(* IEC 61131-3 sources: iec-checker/test/st, 51 files *)

(* ---- declaration-analysis.st ---- *)
(* This demo includes some declaration errors *)
TYPE
    (* String types *)
    ST0 : STRING[5];                               (* OK *)
    ST1 : STRING;                                  (* OK *)
    ST2 : STRING[5] := 'foo';                      (* OK *)
    ST3 : STRING := 'platform_dependent';          (* OK *)
    ST4 : STRING[5] := "foobar";                   (* Error *)

    (* Subrange types *)
    ANALOG_DATA1 : INT (-4095 .. 4095);          (* OK *)
    ANALOG_DATA1 : INT (-4095 .. 4095) := 2000;  (* OK *)
    ANALOG_DATA1 : INT (-4095 .. 4095) := 4095;  (* OK: See 6.4.4.4.1 *)
    ANALOG_DATA1 : INT (-4095 .. 4095) := -4095; (* OK: See 6.4.4.4.1 *)
    ANALOG_DATA2 : INT (-4095 .. 4095) := 4099;  (* Error *)
    ANALOG_DATA2 : INT (-4095 .. 4095) := -4096; (* Error *)
END_TYPE

(* ---- merge-1.st ---- *)
TYPE example_struct :
  STRUCT
    Field : BOOL;
  END_STRUCT
END_TYPE

(* ---- plcopen-cp13.st ---- *)
(* Uncompatible: Recursive functions are forbidden *)
FUNCTION Factorial : INT
    VAR_INPUT
        X : INT;
    END_VAR

    IF X > 1 THEN
        Factorial := Factorial(X - 1) * X;
    ELSE
        Factorial := X;
    END_IF;
END_FUNCTION

(* Compatible iterative implementation *)
FUNCTION Factorial_good : INT
    VAR_INPUT
        X : INT;
    END_VAR
    VAR
        Acc : INT;
    END_VAR

    FOR I := 0 TO 100 DO
        Acc := Acc * X;
    END_FOR;
    Factorial := Acc;
END_FUNCTION

(* ---- plcopen-cp4.st ---- *)
FUNCTION demo : INT
    VAR_INPUT
        x1 AT %MX40 : INT; (* PLCOPEN-CP4 *)
        x2 AT %MX41 : INT; (* PLCOPEN-CP4 *)
        x3 AT %MX510 : INT;
        w1 AT %MW10 : INT; (* adjacent words don't overlap *)
        w2 AT %MW11 : INT;
        d1 AT %MW20 : DINT; (* PLCOPEN-CP4 *)
        d2 AT %MW21 : INT; (* PLCOPEN-CP4 *)
        b1 AT %MB30 : INT; (* PLCOPEN-CP4 *)
        b2 AT %MB31 : BYTE; (* PLCOPEN-CP4 *)
        i1 AT %IW50 : INT; (* different areas don't overlap *)
        q1 AT %QW50 : INT;
        s1 AT %MW60 : INT; (* PLCOPEN-CP4 *)
        s2 AT %MW60 : INT; (* PLCOPEN-CP4 *)
    END_VAR
    x1 := 42;
END_FUNCTION

(* ---- plcopen-n4.st ---- *)
FUNCTION StartMotor : BOOL
  VAR
    goodVar : INT;
    BadVar  : INT;  (* PLCOPEN-N4 *)
  END_VAR
  StartMotor := TRUE;
END_FUNCTION

FUNCTION start_motor : BOOL    (* PLCOPEN-N4 *)
  start_motor := FALSE;
END_FUNCTION

(* ---- plcopen-n6.st ---- *)
FUNCTION Go : BOOL   (* PLCOPEN-N6 *)
  Go := TRUE;
END_FUNCTION

FUNCTION ReadAndScaleTheTemperatureInput : REAL   (* PLCOPEN-N6 *)
  ReadAndScaleTheTemperatureInput := 0.0;
END_FUNCTION

FUNCTION StartFeeding : BOOL
  StartFeeding := TRUE;
END_FUNCTION

(* ---- comparison.st ---- *)
FUNCTION_BLOCK Example
    VAR_EXTERNAL
        global_var : INT;
    END_VAR
    global_var := 42;
END_FUNCTION_BLOCK

PROGRAM Simple
  VAR_INPUT
    x : TIME;
  END_VAR
  VAR
    temp : DINT;
    i : DINT;
    arr1: ARRAY [1..2] OF BOOL;
    unused_var AT %IW1.2 : REAL := 200.0;
    head AT %B0 : INT;
  END_VAR

  IF i > 10 THEN
    temp := i;
    head := 20;
  END_IF

  WHILE i < 10 DO
    IF i = 5 THEN
      temp := i;
      EXIT;
      i := 42;
    END_IF
    i := i + 1;
  END_WHILE

  ARR1[3] := 19;
  ARR1[2,1] := 19;
  IF x = T#100MS THEN
    %B0 := 42;
  END_IF
END_PROGRAM

(* ---- cross-pou.st ---- *)
(* Programs of one task sharing outputs, globals and FB instances, directly
   and through a function block. See test_cross_pou in test_plcopen.py. *)
CONFIGURATION cfg
  VAR_GLOBAL
    gOut AT %QX2.0 : BOOL;
    gT : TON;
    g2 : INT;
    g3 : pt;
    g4 : BOOL;
    head AT %MW600 : INT;
    gm AT %MW451 : INT;
  END_VAR
  RESOURCE res ON PLC
    TASK fast(INTERVAL := T#10MS, PRIORITY := 1);
    PROGRAM i1 WITH fast : p1;
    PROGRAM i2 WITH fast : p2;
  END_RESOURCE
END_CONFIGURATION

TYPE pt : STRUCT x : INT; END_STRUCT END_TYPE

FUNCTION_BLOCK drv
  VAR_EXTERNAL gOut : BOOL; g2 : INT; gT : TON; END_VAR
  VAR_INPUT v : BOOL; END_VAR
  gOut := v;
  g2 := 1;
  gT(IN := v, PT := T#1S);
END_FUNCTION_BLOCK

PROGRAM p1
  VAR_EXTERNAL gOut : BOOL; gT : TON; g2 : INT; g3 : pt; g4 : BOOL; head : INT; END_VAR
  VAR
    out1 AT %QX0.0 : BOOL;
    r AT %MW450 : REAL;
    b1 AT %IX0.0 : BOOL;
    c : BOOL;
    t : TON;
    tmp : INT;
    d1 : drv;
    cnt : CTU;
    i : INT;
  END_VAR
  out1 := TRUE;
  gOut := c;
  gT(IN := c, PT := T#1S);
  g2 := 2;
  g3.x := 1;
  t(IN := c, PT := T#1S, Q => g4);
  %MW600 := 1;
  tmp := %MW600;
  d1(v := c);
  FOR i := 0 TO 3 DO
    cnt(CU := c);
  END_FOR;
END_PROGRAM

PROGRAM p2
  VAR_EXTERNAL gT : TON; g3 : pt; g4 : BOOL; END_VAR
  VAR
    out2 AT %QX0.0 : BOOL;
    r2 AT %MW450 : INT;
    b2 AT %IX0.0 : BOOL;
    c : BOOL;
    t : TON;
    d2 : drv;
  END_VAR
  out2 := TRUE;
  gT(IN := c, PT := T#1S);
  g3.x := 2;
  t(IN := c, PT := T#1S, Q => g4);
  d2(v := NOT c);
END_PROGRAM

(* ---- dvar.st ---- *)
FUNCTION_BLOCK Example
    VAR_EXTERNAL
        global_var : INT;
    END_VAR
    global_var := 42;
END_FUNCTION_BLOCK

PROGRAM Simple
  VAR
    temp : DINT;
    i : DINT;
    unused_var AT %IW1.2 : REAL := 200.0;
    head AT %B0 : INT;
  END_VAR

  i := head;
  i := 42;
  i := 42 + head;
  i := unused_var + 42;
  i := -head;
  i := Example(head);

END_PROGRAM

(* ---- plcopen-cp12.st ---- *)
CONFIGURATION cfg
  VAR_GLOBAL
    g_valve AT %QX1.0 : BOOL;
  END_VAR
  RESOURCE res ON PLC
    TASK main(INTERVAL := T#10MS, PRIORITY := 1);
    PROGRAM inst WITH main : demo;
  END_RESOURCE
END_CONFIGURATION

FUNCTION_BLOCK act
  VAR_OUTPUT
    out : INT;
  END_VAR
  out := 1;
END_FUNCTION_BLOCK

PROGRAM demo
  VAR_EXTERNAL
    g_valve : BOOL;
  END_VAR
  VAR
    motor AT %QW0 : INT;
    lamps AT %QW10 : WORD;
    temp : INT;
    alarm, run : BOOL;
    i : INT;
    a1 : act;
  END_VAR
  %QW1 := temp;
  IF alarm THEN
    %QW1 := 0; (* PLCOPEN-CP12 *)
  END_IF;
  IF run THEN (* exclusive branches are fine *)
    %QW3 := 1;
  ELSE
    %QW3 := 0;
  END_IF;
  motor := temp;
  %QW0 := 5; (* PLCOPEN-CP12 *)
  lamps.%X0 := TRUE; (* different bits are different outputs *)
  lamps.%X1 := TRUE;
  lamps.%X1 := FALSE; (* PLCOPEN-CP12 *)
  FOR i := 0 TO 3 DO
    %QW4 := i; (* PLCOPEN-CP12 *)
  END_FOR;
  g_valve := run;
  g_valve := alarm; (* PLCOPEN-CP12 *)
  a1(out => %QW5);
  %QW5 := 2; (* PLCOPEN-CP12 *)
  IF run THEN
    %QW6 := 1;
  ELSE
    %QW6 := 0;
  END_IF;
  %QW6 := 2; (* PLCOPEN-CP12 *)
  IF alarm THEN
    %QW7 := 0;
    RETURN;
  END_IF;
  %QW7 := 1; (* not in the same cycle as the write before RETURN *)
  temp := 1; (* not an output *)
  temp := 2;
END_PROGRAM

(* ---- plcopen-cp13-indirect.st ---- *)
FUNCTION fa : INT
  VAR_INPUT x : INT; END_VAR
  fa := fb_(x - 1); (* CP13 *)
END_FUNCTION
FUNCTION fb_ : INT
  VAR_INPUT x : INT; END_VAR
  fb_ := fa(x); (* CP13 *)
END_FUNCTION
FUNCTION fact : INT
  VAR_INPUT x : INT; END_VAR
  fact := MAX(IN1 := fact(x - 1), IN2 := 1); (* CP13 *)
END_FUNCTION
FUNCTION fact3 : INT
  VAR_INPUT x : INT; END_VAR
  fact3 := ABS(fact3(x - 1)); (* CP13 *)
END_FUNCTION
FUNCTION_BLOCK loop_fb
  VAR inner : loop_fb2; END_VAR
  inner(); (* CP13 *)
END_FUNCTION_BLOCK
FUNCTION_BLOCK loop_fb2
  VAR back : loop_fb; END_VAR
  back(); (* CP13 *)
END_FUNCTION_BLOCK
FUNCTION helper : INT
  helper := 1;
END_FUNCTION
FUNCTION user : INT
  user := helper() + helper();
END_FUNCTION

(* ---- plcopen-cp16.st ---- *)
FUNCTION_BLOCK MyFB
  VAR x : INT; END_VAR
  x := 0;
END_FUNCTION_BLOCK

FUNCTION MyFun : INT
  MyFun := 0;
END_FUNCTION

PROGRAM MyProgram
  VAR y : INT; END_VAR
  y := 0;
END_PROGRAM

(* The rule's example, after Figure 20 of IEC 61131-3 *)
PROGRAM F
  VAR_INPUT x1 : BOOL; END_VAR
  VAR_OUTPUT y1 : BOOL; END_VAR
  y1 := x1;
END_PROGRAM

PROGRAM G
  VAR_OUTPUT OUT1 : BYTE; END_VAR
  VAR FB1 : TON; FB2 : TON; END_VAR
  OUT1 := 0;
END_PROGRAM

CONFIGURATION config
  VAR_GLOBAL w : BYTE; END_VAR
  RESOURCE res1 ON PLC
    TASK Fast(INTERVAL := T#10ms, PRIORITY := 1);
    TASK Slow(INTERVAL := T#100ms, PRIORITY := 2);
    PROGRAM inst1 WITH Fast : MyProgram;
    PROGRAM inst2 WITH Slow : MyFB; (* CP16 *)
    PROGRAM inst3 : MyProgram;
    PROGRAM inst4 WITH Fast : MyFun; (* CP16 *)
    PROGRAM inst5 WITH Slow : TON; (* CP16 *)
    PROGRAM inst6 WITH Slow : Unknown;
  END_RESOURCE
  RESOURCE STATION_1 ON PROCESSOR_TYPE_1
    VAR_GLOBAL z1 : BYTE; END_VAR
    TASK SLOW_1(INTERVAL := t#20ms, PRIORITY := 2);
    TASK FAST_1(INTERVAL := t#10ms, PRIORITY := 1);
    PROGRAM P1 WITH SLOW_1 : F(x1 := %IX1.1);
    PROGRAM P2 : G(OUT1 => w,
      FB1 WITH SLOW_1, (* CP16 *)
      FB2 WITH FAST_1); (* CP16 *)
  END_RESOURCE
END_CONFIGURATION

(* ---- plcopen-cp17-members.st ---- *)
TYPE pt : STRUCT x : INT; y : INT; END_STRUCT END_TYPE
FUNCTION_BLOCK f
  VAR_INPUT
    pin : pt;
    other : pt;
  END_VAR
  VAR_OUTPUT
    pout : pt;
    q : INT;
  END_VAR
  pout.x := pin.x;
  other.x := 1;
  q := other.y;
END_FUNCTION_BLOCK

(* ---- plcopen-cp17.st ---- *)
FUNCTION_BLOCK FB_CP17_Test
VAR_INPUT
    in_ok_read_only       : INT;   // Compliant: read at least once, never written
    in_violate_unused     : INT;   // Violation: never read
    in_violate_write_only : INT;   // Violation: written, not read
    in_violate_read_write : INT;   // Violation: read but also written

    idx_read_only           : INT;   // Compliant: only read as array index
    idx_violate_write_only  : INT;   // Violation: written, not read
    func_violate_unused     : INT;   // Violation: never use
    func_read_only          : INT;   // Compliant: only read in func call
    func_violate_write      : INT;   // Violation: written in func call
END_VAR

VAR_OUTPUT
    out_ok_written        : INT;   // Compliant: written at least once
    out_violate_unused    : INT;   // Violation: never written
    out_violate_read_only : INT;   // Violation: read but not written
END_VAR

VAR_IN_OUT
    io_ok_read_only       : INT;   // Compliant: read only
    io_ok_write_only      : INT;   // Compliant: written only
    io_ok_read_write      : INT;   // Compliant: both read and written
    io_violate_unused     : INT;   // Violation: neither read nor written
END_VAR

VAR
    temp : INT;
    arr  : ARRAY[0..9] OF INT;
    func : MYFUNC;
END_VAR

(* ===== VAR_INPUT tests ===== *)

(* Compliant: input parameter is read *)
temp := in_ok_read_only + 1;

(* Violation: in_violate_unused is never used *)

(* Violation: input parameter is written *)
in_violate_write_only := 100;

(* Violation: input parameter is both read and written *)
temp := in_violate_read_write;
in_violate_read_write := temp + 1;

(* ===== VAR_OUTPUT tests ===== *)

(* Compliant: output parameter is written *)
out_ok_written := temp;

(* Violation: out_violate_unused is never written *)

(* Violation: output parameter is read but not written *)
temp := out_violate_read_only;

(* ===== VAR_IN_OUT tests ===== *)

(* Compliant: read only *)
temp := temp + io_ok_read_only;

(* Compliant: written only *)
io_ok_write_only := 10;

(* Compliant: both read and written *)
io_ok_read_write := io_ok_read_write + 1;

(* Violation: io_violate_unused is never used *)

(* ===== special tests for LHS handling ===== *)

(* Important case:
   idx_read_only is used only to locate the write target arr[idx_read_only].
   It should be counted as READ, not WRITE.
   However, *)
arr[idx_read_only] := 5;

(* Violation:
   idx_violate_write_only is written, but never read. *)
idx_violate_write_only := 3;

(* Function Call *)
func(func_violate_unused := func_read_only, func_violate_unused => func_violate_write);

END_FUNCTION_BLOCK

(*
 * The reported result should be:
 * 1. in_violate_unused => should be read
 * 2. in_violate_write_only => should not be written, should be read (2 * warnings reported)
 * 3. in_violate_read_write => should not be written
 * 4. out_violate_unused => should be written
 * 5. out_violate_read_only => should be written
 * 6. io_violate_unused => should be written/read
 * 7. idx_violate_write_only => should not be written, should be read (2 * warnings reported)
 * 8. func_violate_unused => never used, should be read
 * 9. func_violate_write => should not be written, should be read (2 * warnings reported)
*)

(* ---- plcopen-cp2-library.st ---- *)
(* A library: no program uses these here, but applications do. *)
FUNCTION Scale : INT
  VAR_INPUT x : INT; END_VAR
  Scale := x * 2;
END_FUNCTION

FUNCTION_BLOCK Valve
  VAR_OUTPUT open : BOOL; END_VAR
  open := TRUE;
END_FUNCTION_BLOCK

(* ---- plcopen-cp2-unreferenced.st ---- *)
CONFIGURATION cfg
  VAR_GLOBAL
    g_valve : Valve;
  END_VAR
  RESOURCE res ON PLC
    TASK t (INTERVAL := T#10ms, PRIORITY := 1);
    PROGRAM main_inst WITH t : Main;
  END_RESOURCE
END_CONFIGURATION

FUNCTION Scale : INT
  VAR_INPUT x : INT; END_VAR
  Scale := x * 2;
END_FUNCTION

FUNCTION Clamp : INT
  VAR_INPUT x : INT; END_VAR
  Clamp := x;
END_FUNCTION

FUNCTION Unused : INT (* CP2 *)
  VAR_INPUT x : INT; END_VAR
  Unused := x;
END_FUNCTION

FUNCTION Recurse : INT (* CP2 *)
  VAR_INPUT n : INT; END_VAR
  Recurse := Recurse(n - 1);
END_FUNCTION

FUNCTION OnlyForDeadFb : INT (* CP2 *)
  OnlyForDeadFb := 1;
END_FUNCTION

FUNCTION_BLOCK Valve
  VAR_OUTPUT open : BOOL; END_VAR
  open := TRUE;
END_FUNCTION_BLOCK

FUNCTION_BLOCK Pump
  VAR_OUTPUT running : BOOL; END_VAR
  running := TRUE;
END_FUNCTION_BLOCK

FUNCTION_BLOCK Mixer
  VAR_OUTPUT active : BOOL; END_VAR
  active := TRUE;
END_FUNCTION_BLOCK

FUNCTION_BLOCK DeadFb (* CP2 *)
  VAR_OUTPUT v : INT; END_VAR
  v := OnlyForDeadFb();
END_FUNCTION_BLOCK

TYPE Station :
  STRUCT
    mixer : Mixer;
  END_STRUCT;
END_TYPE

PROGRAM Main
  VAR
    pumps : ARRAY [1..2] OF Pump;
    st : Station;
    y : INT;
  END_VAR
  y := Clamp(Scale(y));
END_PROGRAM

PROGRAM Spare (* CP2 *)
  VAR y : INT; END_VAR
  y := 1;
END_PROGRAM

(* ---- plcopen-cp20.st ---- *)
FUNCTION_BLOCK counter
  VAR_INPUT
    x : BOOL;
  END_VAR
  VAR_OUTPUT
    n : INT;
  END_VAR
  IF x THEN
    n := n + 1;
  END_IF;
END_FUNCTION_BLOCK

FUNCTION helper : INT
  VAR_INPUT
    a : INT;
  END_VAR
  helper := a;
END_FUNCTION

PROGRAM demo
  VAR
    edge1, edge2 : R_TRIG;
    t1 : TON;
    c1 : counter;
    input_a, input_b, run : BOOL;
    i, y : INT;
  END_VAR
  edge1(CLK := input_a);
  edge1(CLK := input_b); (* PLCOPEN-CP20 *)
  edge2(CLK := input_a); (* a different instance *)
  IF run THEN (* exclusive branches are fine *)
    t1(IN := TRUE, PT := T#1S);
  ELSE
    t1(IN := FALSE, PT := T#1S);
  END_IF;
  FOR i := 0 TO 3 DO
    c1(x := run); (* PLCOPEN-CP20 *)
  END_FOR;
  helper(a := 1); (* functions can be called any number of times *)
  helper(a := 2);
  y := helper(3);
END_PROGRAM

(* ---- plcopen-cp25.st ---- *)
TYPE percent : USINT; END_TYPE

TYPE motor_t :
  STRUCT
    speed : DINT;
    temp : REAL;
  END_STRUCT
END_TYPE

FUNCTION_BLOCK sensor
  VAR_INPUT
    limit : INT;
  END_VAR
  VAR_OUTPUT
    value : LREAL;
  END_VAR
  value := 1.0;
END_FUNCTION_BLOCK

FUNCTION scale : DINT
  VAR_INPUT
    x : INT;
    k : REAL;
  END_VAR
  scale := x;
END_FUNCTION

PROGRAM demo
  VAR
    s : SINT;
    I : INT := 10;
    J : REAL := 0.55;
    d : DINT;
    u : UINT;
    lr : LREAL;
    p : percent;
    m : motor_t;
    arr : ARRAY [0..3] OF DINT;
    fb : sensor;
    c : BOOL;
  END_VAR
  (* Conversions without loss are allowed (Table 11) *)
  I := s;
  d := I;
  J := I;
  lr := J;
  c := I < J;
  (* Explicit conversions *)
  I := REAL_TO_INT(J);
  J := INT_TO_REAL(I);
  I := DINT_TO_INT(d);
  (* Lossy implicit conversions *)
  I := J; (* PLCOPEN-CP25 *)
  I := I * J; (* PLCOPEN-CP25 *)
  I := d; (* PLCOPEN-CP25 *)
  I := d + 1; (* PLCOPEN-CP25 *)
  u := I; (* PLCOPEN-CP25 *)
  J := lr; (* PLCOPEN-CP25 *)
  I := 5.7; (* PLCOPEN-CP25 *)
  s := 300; (* PLCOPEN-CP25 *)
  s := 100;
  u := -1; (* PLCOPEN-CP25 *)
  p := I; (* PLCOPEN-CP25 *)
  I := m.speed; (* PLCOPEN-CP25 *)
  I := arr[1]; (* PLCOPEN-CP25 *)
  J := fb.value; (* PLCOPEN-CP25 *)
  I := scale(I, J); (* PLCOPEN-CP25 *)
  I := %IW0; (* PLCOPEN-CP25 *)
  d := %IW0;
  (* Operands without a lossless common type *)
  c := d < J; (* PLCOPEN-CP25 *)
  c := I = u; (* PLCOPEN-CP25 *)
  (* Arguments *)
  fb(limit := d); (* PLCOPEN-CP25 *)
  fb(limit := I);
  d := scale(d, J); (* PLCOPEN-CP25 *)
  d := scale(x := I, k := lr); (* PLCOPEN-CP25 *)
END_PROGRAM

(* ---- plcopen-cp28.st ---- *)
PROGRAM demo
    VAR
        x : TIME;
        y : TIME;
        t1 : TON;
        now, shift_start : TOD;
        today, due : DATE;
        ready, b : BOOL;
    END_VAR

    IF x = T#100MS THEN (* PLCOPEN CP-28 *)
      x := x + 1;
    END_IF;

    IF x <> T#100MS THEN (* PLCOPEN CP-28 *)
      x := x + 1;
    END_IF;

    IF T#100MS = x THEN (* PLCOPEN CP-28 *)
      x := x + 1;
    END_IF;

    IF T#100MS <> x THEN (* PLCOPEN CP-28 *)
      x := x + 1;
    END_IF;

    IF REAL_TO_INT(x) <> 0 THEN (* PLCOPEN CP-28: a time in an integer *)
      x := x + 1;
    END_IF;

    IF x = y THEN (* PLCOPEN CP-28 *)
      x := T#0S;
    END_IF;
    IF t1.ET = x THEN (* PLCOPEN CP-28 *)
      x := T#0S;
    END_IF;
    b := ready AND x <> y; (* PLCOPEN CP-28 *)
    IF now = shift_start THEN (* PLCOPEN CP-28 *)
      x := T#0S;
    END_IF;
    IF today = due THEN (* dates can be compared for equality *)
      x := T#0S;
    END_IF;
    IF t1.ET >= x THEN (* ordering comparisons are fine *)
      x := T#0S;
    END_IF;
    IF today = D#2024-01-01 THEN (* date literals are dates *)
      x := T#0S;
    END_IF;
    IF now = TOD#08:00:00 THEN (* PLCOPEN CP-28 *)
      x := T#0S;
    END_IF;
END_PROGRAM

FUNCTION_BLOCK Stopwatch
    VAR_INPUT run : BOOL; END_VAR
    VAR_OUTPUT elapsed_ms : DINT; count : INT; END_VAR
    VAR t : TON; END_VAR
    t(IN := run, PT := T#1H);
    elapsed_ms := TIME_TO_DINT(t.ET);
    count := count + 1;
END_FUNCTION_BLOCK

FUNCTION SecondsOf : DINT
    VAR_INPUT d : TIME; END_VAR
    SecondsOf := TIME_TO_DINT(d) / 1000;
END_FUNCTION

PROGRAM integers
    VAR
        t1 : TON;
        sw : Stopwatch;
        ms, secs, n, code : DINT;
        r : REAL;
    END_VAR
    (* The rule's example: a time in integer format. *)
    IF TIME_TO_DINT(t1.ET) = 10000 THEN (* PLCOPEN CP-28 *)
      n := 0;
    END_IF;
    ms := TIME_TO_DINT(t1.ET);
    secs := ms / 1000;
    IF secs = 10 THEN (* PLCOPEN CP-28 *)
      n := 0;
    END_IF;
    IF TO_DINT(t1.ET) <> ms THEN (* PLCOPEN CP-28 *)
      n := 0;
    END_IF;
    IF sw.elapsed_ms = 500 THEN (* PLCOPEN CP-28 *)
      n := 0;
    END_IF;
    IF SecondsOf(t1.ET) = 3 THEN (* PLCOPEN CP-28 *)
      n := 0;
    END_IF;
    IF ms > 10000 THEN (* ordering comparisons are fine *)
      n := 0;
    END_IF;
    IF sw.count = 3 OR code = 7 THEN (* other integers are fine *)
      n := 0;
    END_IF;
    r := TIME_TO_REAL(t1.ET);
    IF n = 0 THEN
      n := 1;
    END_IF;
END_PROGRAM

(* ---- plcopen-cp6-constants.st ---- *)
CONFIGURATION cfg
  VAR_GLOBAL CONSTANT
    MAX_SPEED : INT := 1500;
  END_VAR
  VAR_GLOBAL
    ModeAuto : BOOL;
  END_VAR
END_CONFIGURATION

FUNCTION_BLOCK motor
  VAR_EXTERNAL CONSTANT
    MAX_SPEED : INT;
  END_VAR
  VAR_EXTERNAL
    ModeAuto : BOOL; (* CP6 *)
  END_VAR
  VAR_OUTPUT q : BOOL; END_VAR
  q := ModeAuto AND MAX_SPEED > 0;
END_FUNCTION_BLOCK

FUNCTION limit_of : INT
  VAR_EXTERNAL
    MAX_SPEED : INT; (* references a constant global *)
  END_VAR
  limit_of := MAX_SPEED;
END_FUNCTION

(* ---- plcopen-cp6.st ---- *)
FUNCTION demo : INT
    VAR_EXTERNAL
        x1 : INT; (* PLCOPEN-CP6 *)
    END_VAR
    x1 := 42;
END_FUNCTION

FUNCTION_BLOCK demo
    VAR_EXTERNAL
        x1 : INT; (* PLCOPEN-CP6 *)
    END_VAR
    x1 := 42;
END_FUNCTION_BLOCK

PROGRAM demo
    VAR_EXTERNAL
        x1 : INT;
    END_VAR
    x1 := 42;
END_PROGRAM

CLASS test1
  VAR_EXTERNAL
    x1 : INT; (* PLCOPEN-CP6 *)
  END_VAR

  METHOD PRIVATE count
    x1 := 42;
  END_METHOD

END_CLASS

(* ---- plcopen-cp7.st ---- *)
FUNCTION_BLOCK Scaler
  VAR_INPUT P1 : INT; P2 : INT; END_VAR
  VAR_OUTPUT Out : INT; xError : BOOL; iError : INT; END_VAR
  Out := P1 * P2;
  xError := FALSE;
  iError := 0;
END_FUNCTION_BLOCK

FUNCTION ReadSensor : INT
  VAR_INPUT channel : INT; END_VAR
  VAR_OUTPUT ErrorCode : INT; END_VAR
  ReadSensor := channel;
  ErrorCode := 0;
END_FUNCTION

FUNCTION_BLOCK Wrapper
  VAR_OUTPUT xError : BOOL; END_VAR
  VAR inner : Scaler; END_VAR
  inner(P1 := 1, P2 := 2, xError => xError);   (* passed on as its own output *)
END_FUNCTION_BLOCK

PROGRAM Main
  VAR
    Cond : BOOL;
    Eff1 : INT;
    Eff2 : INT;
    Result : INT;
    CriticalThreshold : INT;
    instance : Scaler;
    checked : Scaler;
    connected : Scaler;
    ignored : Scaler;
    err : BOOL;
    code : INT;
    unread : INT;
    unreadFlag : BOOL;
    value : INT;
    move : MC_MoveAbsolute;
    power : MC_Power;
    wrap : Wrapper;
  END_VAR
  (* The rule's example: Result is used without checking the error *)
  instance(P1 := Eff1, P2 := Eff2);   (* PLCOPEN-CP7 *)
  Result := instance.Out;
  CriticalThreshold := Result + 10000;

  (* Tested: read directly, or connected and read *)
  checked(P1 := Eff1, P2 := Eff2);
  IF NOT checked.xError AND checked.iError = 0 THEN
    CriticalThreshold := checked.Out + 10000;
  END_IF;
  connected(P1 := Eff1, P2 := Eff2, xError => err, iError => code);
  IF NOT err AND code = 0 THEN
    Result := connected.Out;
  END_IF;
  ignored(P1 := 1, P2 := 2, xError => unreadFlag, iError => unread);   (* PLCOPEN-CP7 *)

  (* Functions with an error output *)
  value := ReadSensor(channel := 1, ErrorCode => code);
  value := ReadSensor(channel := 2);   (* PLCOPEN-CP7 *)
  unread := ReadSensor(channel := 3, ErrorCode => unread);   (* PLCOPEN-CP7 *)

  (* Motion control blocks *)
  move(Execute := Cond);   (* PLCOPEN-CP7 *)
  power(Enable := TRUE);
  IF power.Error THEN
    Cond := FALSE;
  END_IF;   (* testing Error is enough *)

  (* The error of wrap is passed on as its own output *)
  wrap();
  Cond := wrap.xError;
END_PROGRAM

(* ---- plcopen-cp9.st ---- *)
(* Example from PLCOpen guidelines, page 60.

   The following Function block CHARCURVE has:
   Number of Statements 18
   McCabe complexity of 12
   Prater complexity of 3,89
   Halstead complexity of 44,9
   Elshof complexity of 0,14

  Counting each statement once, including ELSIF but not ELSE, gives their 18
  statements. Their McCabe value comes out with the "plcopen" variant; the
  standard McCabe complexity is 8. CHARCURVE2 is the improved version of the
  rule's example: 12 statements, and McCabe complexity 8 (standard: 6).
 *)

FUNCTION_BLOCK CHARCURVE
  VAR_INPUT
    IN:INT;
    N:BYTE;
  END_VAR
  (* VAR_IN_OUT *)
    (* P : ARRAY [0 .. 10] OF POINT; *)
  (* END_VAR *)
  VAR_OUTPUT
    OUT:INT;
    ERR: BYTE;
  END_VAR
  VAR
    I:INT;
  END_VAR

  IF N > 1 AND N < 12 THEN
    ERR:=0;
    (* IF IN < P[0].X THEN *)
    IF IN < a THEN
      ERR := 2;
      OUT := DINT_TO_INT(a);
    (* ELSIF IN > P[N-1].X THEN *)
    ELSIF IN > a THEN
      ERR := 2;
      OUT := DINT_TO_INT(a);
    ELSE
      FOR I:=1 TO N-1 DO
        (* IF P[I-1].X >= P[I].X THEN *)
        IF a >= a THEN
          ERR:=1;
          EXIT;
        END_IF;
        (* IF IN <= P[I].X THEN *)
        IF IN <= a THEN
          EXIT;
        END_IF;
      END_FOR;
      IF ERR = 0 THEN
        (* OUT := DINT_TO_INT(P[I].Y - (P[I].X-IN) * (P[I].Y-P[I-1].Y) / (P[I].X-P[I-1].X)); *)
        OUT := DINT_TO_INT(a - (a - IN) * (a - a) / (a - a));
      ELSE
        OUT:=0;
      END_IF;
    END_IF;
  ELSE
    ERR := 4;
  END_IF;
END_FUNCTION_BLOCK

FUNCTION_BLOCK CHARCURVE2
  VAR_INPUT
    IN:INT;
    N:BYTE;
  END_VAR
  VAR_OUTPUT
    OUT:INT;
    ERR: BYTE;
  END_VAR
  VAR
    I:INT;
    iIndexFound:INT;
  END_VAR

  OUT := 0;
  ERR := 0;
  iIndexFound := -1;
  FOR I := 1 TO N-1 DO
    (* IF iIndexFound < 0 AND ERR = 0 THEN *)
    IF iIndexFound < 0 AND ERR = 0 THEN
      (* IF P[I-1].X >= P[I].X THEN *)
      IF a >= a THEN
        ERR := 1;
      (* ELSIF IN <= P[I].X THEN *)
      ELSIF IN <= a THEN
        iIndexFound := I;
      END_IF;
    END_IF;
  END_FOR;
  IF ERR = 0 THEN
    (* OUT := CalculateOut(P[iIndexFound], P[iIndexFound - 1]); *)
    OUT := a;
  ELSE
    OUT := 0;
  END_IF;
END_FUNCTION_BLOCK

(* ---- plcopen-l22.st ---- *)
FUNCTION_BLOCK Stepper
  VAR_INPUT step : INT; END_VAR
  VAR_IN_OUT pos : INT; END_VAR
  VAR_OUTPUT next : INT; END_VAR
  pos := pos + step;
  next := pos;
END_FUNCTION_BLOCK

FUNCTION Bump : INT
  VAR_IN_OUT x : INT; END_VAR
  x := x + 1;
  Bump := x;
END_FUNCTION

PROGRAM l22
  VAR
    i : INT := 0;
    j : INT := 0;
    n : INT := 10;
    k : INT := 1;
    arr : ARRAY[0..10] OF INT;
    cfg : Limits;
    st : Stepper;
  END_VAR

  (* Case 1: Direct assignment in body — violation *)
  FOR i := 0 TO 10 BY 2 DO
    IF arr[i] = 42 THEN
      i := 10; (* L22 *)
    END_IF;
  END_FOR;

  (* Case 2: No violation — different variable *)
  FOR i := 0 TO 10 DO
    j := i + 1;
  END_FOR;

  (* Case 3: Nested FOR — inner loop modifies outer var — violation *)
  FOR i := 0 TO 10 DO
    FOR j := 0 TO 5 DO
      i := j; (* L22 *)
    END_FOR;
  END_FOR;

  (* Case 4: Nested FOR — inner loop modifies its own var — violation *)
  FOR i := 0 TO 10 DO
    FOR j := 0 TO 5 DO
      j := 0; (* L22 *)
    END_FOR;
  END_FOR;

  (* Case 5: Nested FOR reuses the outer control variable *)
  FOR i := 0 TO 10 DO
    FOR i := 0 TO 5 DO (* L22 *)
      j := i;
    END_FOR;
  END_FOR;

  (* Case 6: Written through an output and a VAR_IN_OUT *)
  FOR i := 0 TO 10 DO
    st(step := 1, pos := i, next => j); (* L22 *)
  END_FOR;
  FOR j := 0 TO 10 DO
    st(step := 1, pos := k, next => j); (* L22 *)
  END_FOR;
  FOR i := 0 TO 10 DO
    j := Bump(i); (* L22 *)
  END_FOR;

  (* Case 7: The final value and increment change *)
  FOR i := 0 TO n BY k DO
    n := n - 1; (* L22 *)
    k := 2; (* L22 *)
  END_FOR;
  FOR i := 0 TO cfg.max DO
    cfg.max := 5; (* L22 *)
    cfg.min := 1;
  END_FOR;
  FOR i := 0 TO arr[j] DO
    j := j + 1; (* L22 *)
  END_FOR;

  (* Case 8: The initial value is evaluated once *)
  FOR i := j TO 10 DO
    j := 0;
  END_FOR;
END_PROGRAM

(* ---- plcopen-n10-kinds.st ---- *)
TYPE EColor : (Red, Green); END_TYPE
TYPE Error : (Minor, Major); END_TYPE   (* PLCOPEN-N10 *)
TYPE EN_Level : INT (Low := 1, High := 2); END_TYPE
TYPE ELevel : INT (Low2 := 1, High2 := 2); END_TYPE   (* PLCOPEN-N10 *)
TYPE STPoint : STRUCT x : INT; END_STRUCT; END_TYPE
TYPE T_Speed : REAL; END_TYPE
TYPE Speed2 : REAL; END_TYPE   (* PLCOPEN-N10 *)

FUNCTION FUScale : INT
  FUScale := 1;
END_FUNCTION

FUNCTION Scale : INT   (* PLCOPEN-N10 *)
  Scale := 1;
END_FUNCTION

FUNCTION_BLOCK FBPump
  VAR x : INT; END_VAR
  x := 1;
END_FUNCTION_BLOCK

FUNCTION_BLOCK FBpump2   (* PLCOPEN-N10 *)
  VAR x : INT; END_VAR
  x := 1;
END_FUNCTION_BLOCK

PROGRAM PRGMain
  VAR x : INT; END_VAR
  x := 1;
END_PROGRAM

PROGRAM Main   (* PLCOPEN-N10 *)
  VAR x : INT; END_VAR
  x := 1;
END_PROGRAM

(* ---- plcopen-n10.st ---- *)
TYPE
  Color : (Red, Green, Blue);   (* PLCOPEN-N10 *)
END_TYPE

TYPE
  E_Direction : (North, South, East, West);
END_TYPE

FUNCTION_BLOCK Motor   (* PLCOPEN-N10 *)
  VAR
    speed : INT;
  END_VAR
  speed := 0;
END_FUNCTION_BLOCK

FUNCTION_BLOCK FB_Pump
  VAR
    flow : REAL;
  END_VAR
  flow := 0.0;
END_FUNCTION_BLOCK

(* ---- plcopen-n2-scopes.st ---- *)
TYPE Point : STRUCT x : INT; y : INT; END_STRUCT; END_TYPE
TYPE Mode : (Auto, Manual); END_TYPE
TYPE Temperature : REAL; END_TYPE
TYPE Counter : INT; END_TYPE

FUNCTION_BLOCK Pump
  VAR_INPUT
    pxEnable : BOOL;
    xEnable : BOOL;         (* PLCOPEN-N2 *)
  END_VAR
  VAR_OUTPUT
    piCount : INT;
  END_VAR
  VAR
    xReady : BOOL;
    x_done : BOOL;
    xylophone : BOOL;       (* PLCOPEN-N2 *)
    index : INT;            (* PLCOPEN-N2 *)
    todStart : TIME_OF_DAY;
    todEnd : TOD;
    StartAt : TOD;          (* PLCOPEN-N2 *)
    aValues : ARRAY [0..3] OF INT;
    values : ARRAY [0..3] OF INT;  (* PLCOPEN-N2 *)
    stOrigin : Point;
    origin : Point;         (* PLCOPEN-N2 *)
    eMode : Mode;
    mode : Mode;            (* PLCOPEN-N2 *)
    fbTimer : TON;
    timer : TON;            (* PLCOPEN-N2 *)
    tempOven : Temperature;
    oven : Temperature;     (* PLCOPEN-N2 *)
    iTotal : Counter;
    total : Counter;        (* PLCOPEN-N2 *)
    unknown : SomeType;
  END_VAR
  xReady := pxEnable;
END_FUNCTION_BLOCK

PROGRAM Main
  VAR xOn : BOOL; END_VAR
  xOn := TRUE;
END_PROGRAM

CONFIGURATION cfg
  VAR_GLOBAL
    gxRunning : BOOL;
    xStopped : BOOL;        (* PLCOPEN-N2 *)
    gCount : INT;           (* PLCOPEN-N2 *)
  END_VAR
  RESOURCE res ON PLC
    VAR_GLOBAL
      giLevel : INT;
      level : INT;          (* PLCOPEN-N2 *)
    END_VAR
    TASK main(INTERVAL := T#10ms, PRIORITY := 1);
    PROGRAM inst WITH main : Main;
  END_RESOURCE
END_CONFIGURATION

(* ---- plcopen-n3-names.st ---- *)
TYPE MAX : STRUCT TP : INT; y : INT; END_STRUCT END_TYPE
TYPE mode : (SEL, RUNNING); END_TYPE
FUNCTION_BLOCK TON2
VAR LEFT, LIMIT, LOG, LE, Temp : INT; END_VAR
LEFT := 1;
END_FUNCTION_BLOCK
FUNCTION LEN : INT
LEN := 1;
END_FUNCTION
PROGRAM CTUD
VAR x : INT; END_VAR
x := 1;
END_PROGRAM

(* ---- plcopen-n5-scopes.st ---- *)
CONFIGURATION cfg
  VAR_GLOBAL
    MyCalculation : REAL;
  END_VAR
  RESOURCE res ON PLC
    VAR_GLOBAL
      ResGlobal : INT;
    END_VAR
    TASK task0(INTERVAL := T#20ms, PRIORITY := 0);
    PROGRAM instance0 WITH task0 : prog0;
  END_RESOURCE
END_CONFIGURATION

PROGRAM prog0
  VAR_EXTERNAL
    MyCalculation : REAL; (* refers to the global *)
  END_VAR
  VAR
    ResGlobal : INT; (* N5 *)
    task0 : INT; (* N5 *)
  END_VAR
  MyCalculation := 1.0;
END_PROGRAM

FUNCTION_BLOCK Example
  VAR
    MyCalculation : REAL; (* N5 *)
  END_VAR
  MyCalculation := 0.0;
END_FUNCTION_BLOCK

(* ---- plcopen-n5.st ---- *)
PROGRAM prog0
  VAR
    local0 : INT;
  END_VAR
  local0 := 0;
END_PROGRAM

FUNCTION_BLOCK Example
  VAR
    MyCalculation : REAL;   (* PLCOPEN-N5 *)
  END_VAR
  MyCalculation := 0.0;
END_FUNCTION_BLOCK

CONFIGURATION config
  VAR_GLOBAL
    MyCalculation : REAL;
  END_VAR
  TASK task0(INTERVAL := T#20ms, PRIORITY := 0);
  PROGRAM instance0 WITH task0 : prog0;
END_CONFIGURATION

(* ---- plcopen-n6-locals.st ---- *)
FUNCTION_BLOCK FeedControl
  VAR_INPUT
    enable : BOOL;   (* PLCOPEN-N6 *)
    startRequest : BOOL;
  END_VAR
  VAR
    i : INT;
    j : INT;   (* PLCOPEN-N6 *)
    sum : INT;
    MaximumTemperatureForTheThermocoupleInput : REAL;   (* PLCOPEN-N6 *)
  END_VAR
  FOR i := 1 TO 10 DO
    sum := sum + i;
  END_FOR;
  j := sum;
END_FUNCTION_BLOCK

FUNCTION Go : BOOL   (* PLCOPEN-N6 *)
  Go := TRUE;
END_FUNCTION

PROGRAM MainProgram
  VAR ctl : FeedControl; END_VAR
  ctl(enable := TRUE);
END_PROGRAM

CONFIGURATION PlantConfig
  VAR_GLOBAL
    speed : INT;   (* PLCOPEN-N6 *)
    conveyorSpeed : INT;
  END_VAR
  RESOURCE res ON PLC
    VAR_GLOBAL
      level : INT;   (* PLCOPEN-N6 *)
    END_VAR
    TASK fast(INTERVAL := T#10ms, PRIORITY := 1);   (* PLCOPEN-N6 *)
    TASK SlowCycle(INTERVAL := T#100ms, PRIORITY := 2);
    PROGRAM mainInst WITH SlowCycle : MainProgram;
  END_RESOURCE
END_CONFIGURATION

(* ---- plcopen-n8.st ---- *)
(* Autorise le départ du wagonnet: accents in comments are fine *)
TYPE Mode : (Automatique, Arrêt); END_TYPE   (* PLCOPEN-N8 *)
TYPE Point : STRUCT x : INT; hauteur_mètres : INT; END_STRUCT; END_TYPE   (* PLCOPEN-N8 *)

FUNCTION_BLOCK Contrôle   (* PLCOPEN-N8 *)
  VAR x : INT; END_VAR
  x := 1;
END_FUNCTION_BLOCK

PROGRAM program0
  VAR
    CleanName : INT;
    another_clean_name : INT;
    départ : BOOL;   (* PLCOPEN-N8 *)
    depart : BOOL;
    double__underscore : INT;   (* PLCOPEN-N8 *)
    trailing_ : INT;   (* PLCOPEN-N8 *)
    _leading : INT;
    変数 : INT;   (* PLCOPEN-N8 *)
  END_VAR
  CleanName := another_clean_name;
  départ := TRUE;
  depart := FALSE;
END_PROGRAM

CONFIGURATION config
  RESOURCE res ON PLC
    TASK tâche(INTERVAL := T#10ms, PRIORITY := 1);   (* PLCOPEN-N8 *)
    PROGRAM instance_ WITH tâche : program0;   (* PLCOPEN-N8 *)
  END_RESOURCE
END_CONFIGURATION

(* ---- plcopen-n9.st ---- *)
PROGRAM prog0   (* PLCOPEN-N9 *)
  VAR
    local0 : INT;
    fast : INT; (* tasks aren't in the scope of POUs *)
  END_VAR
  local0 := 0;
END_PROGRAM

FUNCTION_BLOCK MyCalculation   (* PLCOPEN-N9 *)
  VAR_IN_OUT
    MyCalculation : REAL;   (* PLCOPEN-N9 *)
  END_VAR
  MyCalculation := 1.1;
END_FUNCTION_BLOCK

(* Different kinds of POUs *)
FUNCTION Scale : INT   (* PLCOPEN-N9 *)
  VAR_INPUT x : INT; END_VAR
  Scale := x;
END_FUNCTION

FUNCTION_BLOCK Scale   (* PLCOPEN-N9 *)
  VAR_OUTPUT y : INT; END_VAR
  y := 0;
END_FUNCTION_BLOCK

(* Variables of different POUs don't share a scope *)
FUNCTION_BLOCK Other   (* PLCOPEN-N9 *)
  VAR local0 : INT; END_VAR
  local0 := 1;
END_FUNCTION_BLOCK

CONFIGURATION config
  VAR_GLOBAL
    MyCalculation : REAL;   (* PLCOPEN-N9 *)
    slow : INT;   (* PLCOPEN-N9 *)
  END_VAR
  RESOURCE res ON PLC
    TASK task0(INTERVAL := T#20ms, PRIORITY := 0);
    TASK fast(INTERVAL := T#10ms, PRIORITY := 1);
    TASK slow(INTERVAL := T#100ms, PRIORITY := 2);   (* PLCOPEN-N9 *)
    TASK prog0(INTERVAL := T#50ms, PRIORITY := 3);   (* PLCOPEN-N9 *)
    PROGRAM instance0 WITH task0 : prog0;
    PROGRAM Other WITH fast : prog0;   (* PLCOPEN-N9 *)
  END_RESOURCE
END_CONFIGURATION

(* ---- dead-code.st ---- *)
FUNCTION dead_code_after_return : INT
  VAR
    counter : INT := 0;
    some_var : INT;
  END_VAR
  counter := counter + 1;
  counter := 2 + 2;
  RETURN;
  some_var := SQRT(16#42); (* UnreachableCode error *)
  some_var := 16#42; (* No additional warnings *)
  some_var := 19;
END_FUNCTION

PROGRAM dead_code_in_the_loops
VAR a : INT; i : INT; END_VAR
  WHILE i < 10 DO
    IF i = 5 THEN
      i := i + 1;
      EXIT;
      i := 19; (* UnreachableCode error *)
      i := 42; (* No additional warnings *)
      i := 42;
    ELSIF i = 6 THEN
      CONTINUE;
      i := 3; (* UnreachableCode error *)
      i := 44; (* No additional warnings *)
      i := 19;
    END_IF;
    i := i + 2;
  END_WHILE;
  I := 0;
END_PROGRAM

(* ---- merge-2.st ---- *)
PROGRAM Program1
  VAR
    instance AT %MW500 : example_struct;
  END_VAR

  %MW500 := TRUE;
END_PROGRAM

(* ---- mixed-type-arithmetic.st ---- *)
PROGRAM demo
  VAR
    i : INT;
    d : DINT;
    r : REAL;
    lr : LREAL;
    w : WORD;
    t : TIME;
  END_VAR
  d := i + d; (* MixedTypeArithmetic *)
  r := r * i; (* MixedTypeArithmetic *)
  r := i * 1.5; (* MixedTypeArithmetic *)
  r := r * 2; (* integer literals take the other operand's type *)
  i := i + 1;
  lr := lr + r; (* MixedTypeArithmetic *)
  r := INT_TO_REAL(i) * r; (* explicit conversion *)
  t := t * 2; (* TIME arithmetic isn't numeric *)
  i := i + w; (* MixedTypeArithmetic *)
END_PROGRAM

(* ---- nested-exprs.st ---- *)
PROGRAM p
  VAR
    x : REAL;
    t : TIME;
    y : INT;
  END_VAR

  IF y > 0 THEN
    IF x = 1.5 THEN (* PLCOPEN-CP8 *)
      y := 1;
    END_IF;
    WHILE t = T#1S DO (* PLCOPEN-CP28 *)
      y := 2;
    END_WHILE;
    %QW1 := 3; (* PLCOPEN-N1 *)
  END_IF;
  y := MAX(%MW1, 0); (* PLCOPEN-N1 *)
END_PROGRAM

(* ---- plcopen-cp1.st ---- *)
(** PLCOPEN-CP1 – Access to a member shall be by name *)

PROGRAM program0
  VAR
    head AT %B0 : INT;
  END_VAR
  %B0 := 42;
END_PROGRAM

(* ---- plcopen-cp2.st ---- *)
FUNCTION f1 : INT
  VAR i : INT; END_VAR
  RETURN;
  WHILE i < 10 DO (* CP2 *)
    i := i + 1;
  END_WHILE;
END_FUNCTION

FUNCTION f2 : INT
  VAR c : BOOL; i : INT; END_VAR
  IF c THEN
    RETURN;
  ELSE
    RETURN;
  END_IF;
  i := 1; (* CP2 *)
END_FUNCTION

PROGRAM p
  VAR c : BOOL; i : INT; END_VAR
  IF FALSE THEN (* bypass idiom of the rule *)
    i := 1;
  END_IF;
  IF 1 > 2 THEN
    i := 2; (* CP2 *)
  END_IF;
  WHILE FALSE DO
    i := 3; (* CP2 *)
  END_WHILE;
  IF TRUE THEN
    i := 4;
  ELSIF c THEN
    i := 5; (* CP2 *)
  ELSE
    i := 6; (* CP2 *)
  END_IF;
  FOR i := 5 TO 1 DO
    c := TRUE; (* CP2 *)
  END_FOR;
  FOR i := 5 TO 1 BY -1 DO
    c := TRUE;
  END_FOR;
  IF c THEN
    RETURN;
  END_IF;
  i := 7; (* reachable when c is FALSE *)
  REPEAT
    i := i + 1;
    EXIT;
  UNTIL c END_REPEAT;
  i := 8; (* reachable after EXIT *)
END_PROGRAM

(* ---- plcopen-cp26.st ---- *)
CONFIGURATION config
  VAR_GLOBAL
    SharedCounter : INT;
    ReadOnlyVar : INT;
    MultiWriter : INT;
  END_VAR
  TASK task0(INTERVAL := T#20ms, PRIORITY := 0);
  PROGRAM instance0 WITH task0 : Program1;
END_CONFIGURATION

(* Case 1: SharedCounter written by Program1 and Program2 — violation in Program2 *)
PROGRAM Program1
  VAR_EXTERNAL SharedCounter : INT; END_VAR
  VAR_EXTERNAL ReadOnlyVar : INT; END_VAR
  VAR x : INT; END_VAR
  SharedCounter := SharedCounter + 1;
  x := ReadOnlyVar;
END_PROGRAM

PROGRAM Program2
  VAR_EXTERNAL SharedCounter : INT; END_VAR
  VAR_EXTERNAL ReadOnlyVar : INT; END_VAR
  VAR x : INT; END_VAR
  SharedCounter := 0;
  x := ReadOnlyVar;
END_PROGRAM

(* Case 2: MultiWriter written by Program3 and Program4 — violation in Program4 *)
PROGRAM Program3
  VAR_EXTERNAL MultiWriter : INT; END_VAR
  MultiWriter := 1;
END_PROGRAM

PROGRAM Program4
  VAR_EXTERNAL MultiWriter : INT; END_VAR
  MultiWriter := 2;
END_PROGRAM

(* ---- plcopen-cp3.st ---- *)
TYPE TempLimit : REAL := 250.0; END_TYPE
TYPE Plain : STRUCT a : INT; END_STRUCT END_TYPE

FUNCTION f : INT
  VAR_INPUT
    a : INT; (* set by the caller *)
  END_VAR
  VAR
    b : INT;
  END_VAR
  f := a + b; (* PLCOPEN-CP3 *)
END_FUNCTION

PROGRAM Initialization
  VAR
    NumOfRetries : INT := 3;
    StateLastPosition : INT;
    SpeedAverage : REAL;
    Boiler : TempLimit;
    Pipe : Plain;
    Counter : INT;
    Flag : BOOL;
    Both : INT;
    arr : ARRAY [0..3] OF INT;
    i : INT;
    x : INT;
    r : REAL;
    t : TON;
  END_VAR
  VAR RETAIN
    Kept : INT;
  END_VAR
  VAR
    start AT %IX0.0 : BOOL;
  END_VAR
  (* The rule's example: assigned before use *)
  StateLastPosition := 50;
  SpeedAverage := 0.0;
  x := StateLastPosition + NumOfRetries;
  x := Kept; (* RETAIN *)
  IF start THEN (* physical input *)
    Flag := TRUE;
  END_IF;
  x := Counter; (* PLCOPEN-CP3 *)
  Counter := Counter + 1;
  IF Flag THEN (* PLCOPEN-CP3 *)
    Both := 1;
  ELSE
    Both := 2;
  END_IF;
  x := Both; (* assigned in every branch *)
  FOR i := 0 TO 3 DO
    arr[i] := 0;
  END_FOR;
  x := arr[1]; (* the loop runs at least once *)
  x := Pipe.a; (* PLCOPEN-CP3 *)
  t(IN := Flag, PT := T#1S); (* function block instance *)
  r := Boiler; (* type with a default initial value *)
END_PROGRAM

(* ---- plcopen-cp4-sizes.st ---- *)
PROGRAM p
  VAR
    v_lt AT %MW600 : LTIME;
    after_lt AT %MW604 : INT;
    v_ldt AT %MB700 : LDT;
    after_ldt AT %MB708 : BYTE;
    v_dt AT %MB800 : DATE_AND_TIME;
    after_dt1 AT %MB808 : BYTE;
  END_VAR
  after_lt := 1;
END_PROGRAM

(* ---- plcopen-cp8.st ---- *)
TYPE motor_t :
  STRUCT
    temp : REAL;
  END_STRUCT
END_TYPE

FUNCTION avg : REAL
  avg := 1.0;
END_FUNCTION

PROGRAM demo
    VAR
        x : REAL;
        y : REAL;
        lr : LREAL;
        i, j : INT;
        ready, b : BOOL;
        m : motor_t;
    END_VAR

    IF x = 0.0 THEN (* comparing to 0.0 is an exception of the rule *)
      x := x + 1;
    END_IF;

    IF x <> 0.0 THEN
      x := x + 1;
    END_IF;

    IF 0.0 = x THEN
      x := x + 1;
    END_IF;

    IF 0.0 <> x THEN
      x := x + 1;
    END_IF;

    IF REAL_TO_INT(x) <> 0 THEN
      x := x + 1;
    END_IF;

    IF x - y = 0.1 THEN (* PLCOPEN CP-8 *) (* the rule's example *)
      x := 0.0;
    END_IF;
    IF x = y THEN (* PLCOPEN CP-8 *)
      x := 0.0;
    END_IF;
    IF lr <> x THEN (* PLCOPEN CP-8 *)
      x := 0.0;
    END_IF;
    IF x = 0 THEN
      x := 0.0;
    END_IF;
    IF ready AND x = y THEN (* PLCOPEN CP-8 *)
      x := 0.0;
    END_IF;
    IF m.temp = x THEN (* PLCOPEN CP-8 *)
      x := 0.0;
    END_IF;
    IF avg() <> x THEN (* PLCOPEN CP-8 *)
      x := 0.0;
    END_IF;
    b := x = y; (* PLCOPEN CP-8 *)
    IF i = j THEN (* integers can be compared for equality *)
      x := 0.0;
    END_IF;
    IF x > y THEN (* ordering comparisons are fine *)
      x := 0.0;
    END_IF;
END_PROGRAM

(* ---- plcopen-e.st ---- *)
CONFIGURATION cfg
  VAR_GLOBAL g_ptr : POINTER TO INT; END_VAR
  RESOURCE res ON PLC
    TASK t(INTERVAL := T#10ms, PRIORITY := 1);
    PROGRAM inst WITH t : Main;
  END_RESOURCE
END_CONFIGURATION

PROGRAM Main
  VAR_EXTERNAL g_ptr : POINTER TO INT; END_VAR
  VAR
    x : INT;
    y : INT;
    TEMP : INT;
    buf : ARRAY [0..9] OF INT;
    p : POINTER TO INT;
    q : POINTER TO INT;
    r : REF_TO INT;
    s : REF_TO INT;
    addr : DWORD;
    size : DWORD;
    i : INT;
  END_VAR
  (* E1 *)
  p := __NEW(INT, 10);   (* PLCOPEN-E1 *)
  addr := SysMemAlloc(100);   (* PLCOPEN-E1 *)
  __DELETE(p);

  (* E2 *)
  p := ADR(buf);
  p := p + 2;   (* PLCOPEN-E2 *)
  p := ADR(buf) + i * 2 + 4;   (* PLCOPEN-E2 *)
  addr := ADR(buf);
  size := addr - 16;   (* PLCOPEN-E2 *)
  g_ptr := g_ptr + 2;   (* PLCOPEN-E2 *)
  x := buf[i + 1] + p^;   (* values, not addresses *)
  x := p^ + 1;

  (* E3: the rule's example *)
  IF p^ < q^ AND p < q THEN   (* PLCOPEN-E3 *)
    TEMP := p^;
    p^ := q^;
    q^ := TEMP;
  END_IF;
  IF r >= s THEN   (* PLCOPEN-E3 *)
    x := 1;
  END_IF;
  IF addr > ADR(y) THEN   (* PLCOPEN-E3 *)
    x := 1;
  END_IF;
  IF p = q OR r <> NULL OR r = REF(x) THEN   (* equality is allowed *)
    x := 2;
  END_IF;
  IF buf[1] < buf[2] AND i < 3 THEN
    x := 3;
  END_IF;
END_PROGRAM

(* ---- plcopen-l10.st ---- *)
PROGRAM l10
  VAR
    i : INT := 0;
    j : INT := 0;
    flag : INT := 1;
    counter : INT := 0;
  END_VAR

  FOR i := 0 TO 10 DO
    FOR j := 10 TO 100 BY 2 DO
      IF flag THEN
        EXIT; (* PLCOPEN-CP10 *)
      END_IF;
      counter := counter + 1;
      IF j = 10 THEN
        CONTINUE; (* PLCOPEN-CP10 *)
      END_IF;
      EXIT; (* PLCOPEN-CP10 *)
    END_FOR;
  END_FOR;
END_PROGRAM

(* ---- plcopen-l13.st ---- *)
PROGRAM l13
  VAR
    i : INT := 0;
    j : INT := 0;
    x : INT := 0;
    WORDS : ARRAY[0..100] OF STRING;
    value : STRING := 'val';
  END_VAR

  (* Case 1: Use after FOR — 2 violations *)
  FOR i := 0 TO 100 BY 2 DO
    IF WORDS[i] = 'Key' THEN EXIT; END_IF;
  END_FOR;
  IF i <= 100 THEN
    WORDS[i + 1] := value;
  END_IF;

  (* Case 2: No violation — variable not used after loop *)
  FOR j := 0 TO 10 DO
    x := j;
  END_FOR;

  (* Case 3: Reuse as control var in subsequent FOR — no violation *)
  FOR i := 0 TO 10 DO
    x := i;
  END_FOR;
  FOR i := 0 TO 20 DO
    x := i;
  END_FOR;

  (* Case 4: Nested FOR — outer var used after inner loop — violation *)
  FOR i := 0 TO 10 DO
    FOR j := 0 TO 5 DO
      x := j;
    END_FOR;
    x := j;
  END_FOR;

  (* Case 5: Use in expression after FOR — violation *)
  FOR j := 0 TO 10 DO
    x := j;
  END_FOR;
  x := j + 1;
END_PROGRAM

(* ---- plcopen-l17.st ---- *)
(** PLCOPEN-L17 – Each IF instruction should have an ELSE clause

    Reference: PLCopen Coding Guidelines 6.5.9. *)

PROGRAM program0
  VAR
    a : INT;
  END_VAR

  IF (a = 42) (* PLCOPEN-L17 *)
    THEN
      a := 0;
  END_IF;

  IF (a = 42) (* no warning *)
    THEN
      a := 0;
    ELSE
      a := 19;
  END_IF;

END_PROGRAM

(* ---- plcopen-n1.st ---- *)
PROGRAM l10
  VAR
    a AT %MW10.2.4.1 : INT;
  END_VAR

   %MW10.2.4.1 := 42; (* PLCOPEN-N1 *)
   a := 42; (* ok *)
END_PROGRAM

(* ---- plcopen-n2.st ---- *)
PROGRAM program0
  VAR
    iCounter : INT;
    Counter  : INT;   (* PLCOPEN-N2 *)
    xReady   : BOOL;
    Ready    : BOOL;  (* PLCOPEN-N2 *)
  END_VAR

  iCounter := Counter;
  xReady := Ready;
END_PROGRAM

(* ---- plcopen-n3.st ---- *)
PROGRAM program0
  VAR
    FOR_B : INT; (* starts with a keyword, but isn't one *)
    NO_FALSE_POSITIVE : INT;
    IF_A : INT;
    TOF : INT; (* PLCOPEN-N3 *)
    OK_ALLOWED : INT;
  END_VAR

  FOR_B := IF_A / 1;
END_PROGRAM

(* ---- plcopen-n4-members.st ---- *)
(* The rule's example of structured types *)
TYPE
  ANALOG_SIGNAL_RANGE : (BIPOLAR_10V, unipolar10V);   (* PLCOPEN-N4 *)
END_TYPE
TYPE
  ANALOG_CHANNEL_CONFIGURATION :
    STRUCT
      range : ANALOG_SIGNAL_RANGE;
      MIN_SCALE : INT;   (* PLCOPEN-N4 *)
      maxScale : INT;
    END_STRUCT;
END_TYPE

TYPE MODE : (AUTO_MODE, manualMode); END_TYPE   (* PLCOPEN-N4 *)

FUNCTION StartMotor : BOOL
  StartMotor := TRUE;
END_FUNCTION

FUNCTION STARTMOTOR2 : BOOL   (* PLCOPEN-N4 *)
  STARTMOTOR2 := TRUE;
END_FUNCTION

FUNCTION IO : BOOL
  IO := TRUE;
END_FUNCTION

PROGRAM Main
  VAR
    mode : MODE;
  END_VAR
  VAR CONSTANT
    MAX_SPEED : INT := 100;
    minSpeed : INT := 1;   (* PLCOPEN-N4 *)
  END_VAR
  mode := AUTO_MODE;
END_PROGRAM
